FUNCTION_BLOCK MotorWorkTime
VAR_INPUT
END_VAR
VAR_OUTPUT
END_VAR
VAR
END_VAR

END_FUNCTION_BLOCK

(* stored: Version 1.1.0.1, ProductVersion 3.1.4024.12
   POU MotorWorkTime: Id {bf300658-67ee-4a5c-88df-962f2b07572d}, SpecialFunc None *)
